FUNCTION_BLOCK ASSEMBLE_AL_FROM_AX (* this Function combines the 64 AX (BOOL) adapters to a AL (LWORD) *)
  (* Standard: 61499-2; Description: Copyright (c) 2026 Meisterschulen am Ostbahnhof SPDX-License-Identifier: EPL-2.0 *)
  (* Version 1.0, 2026-05-16, Franz Höpfinger, Meisterschulen am Ostbahnhof, initial API and implementation and/or initial documentation *)
  PACKAGE adapter::assembling;
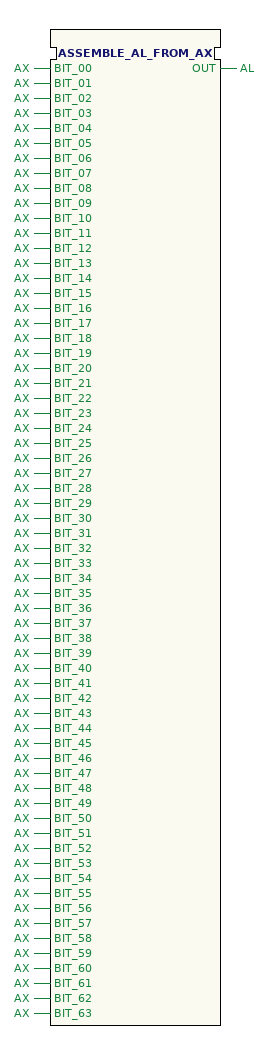
  SOCKETS
    BIT_00 : adapter::types::unidirectional::AX; (* Bool Bit 0 *)
    BIT_01 : adapter::types::unidirectional::AX; (* Bool Bit 1 *)
    BIT_02 : adapter::types::unidirectional::AX; (* Bool Bit 2 *)
    BIT_03 : adapter::types::unidirectional::AX; (* Bool Bit 3 *)
    BIT_04 : adapter::types::unidirectional::AX; (* Bool Bit 4 *)
    BIT_05 : adapter::types::unidirectional::AX; (* Bool Bit 5 *)
    BIT_06 : adapter::types::unidirectional::AX; (* Bool Bit 6 *)
    BIT_07 : adapter::types::unidirectional::AX; (* Bool Bit 7 *)
    BIT_08 : adapter::types::unidirectional::AX; (* Bool Bit 8 *)
    BIT_09 : adapter::types::unidirectional::AX; (* Bool Bit 9 *)
    BIT_10 : adapter::types::unidirectional::AX; (* Bool Bit 10 *)
    BIT_11 : adapter::types::unidirectional::AX; (* Bool Bit 11 *)
    BIT_12 : adapter::types::unidirectional::AX; (* Bool Bit 12 *)
    BIT_13 : adapter::types::unidirectional::AX; (* Bool Bit 13 *)
    BIT_14 : adapter::types::unidirectional::AX; (* Bool Bit 14 *)
    BIT_15 : adapter::types::unidirectional::AX; (* Bool Bit 15 *)
    BIT_16 : adapter::types::unidirectional::AX; (* Bool Bit 16 *)
    BIT_17 : adapter::types::unidirectional::AX; (* Bool Bit 17 *)
    BIT_18 : adapter::types::unidirectional::AX; (* Bool Bit 18 *)
    BIT_19 : adapter::types::unidirectional::AX; (* Bool Bit 19 *)
    BIT_20 : adapter::types::unidirectional::AX; (* Bool Bit 20 *)
    BIT_21 : adapter::types::unidirectional::AX; (* Bool Bit 21 *)
    BIT_22 : adapter::types::unidirectional::AX; (* Bool Bit 22 *)
    BIT_23 : adapter::types::unidirectional::AX; (* Bool Bit 23 *)
    BIT_24 : adapter::types::unidirectional::AX; (* Bool Bit 24 *)
    BIT_25 : adapter::types::unidirectional::AX; (* Bool Bit 25 *)
    BIT_26 : adapter::types::unidirectional::AX; (* Bool Bit 26 *)
    BIT_27 : adapter::types::unidirectional::AX; (* Bool Bit 27 *)
    BIT_28 : adapter::types::unidirectional::AX; (* Bool Bit 28 *)
    BIT_29 : adapter::types::unidirectional::AX; (* Bool Bit 29 *)
    BIT_30 : adapter::types::unidirectional::AX; (* Bool Bit 30 *)
    BIT_31 : adapter::types::unidirectional::AX; (* Bool Bit 31 *)
    BIT_32 : adapter::types::unidirectional::AX; (* Bool Bit 32 *)
    BIT_33 : adapter::types::unidirectional::AX; (* Bool Bit 33 *)
    BIT_34 : adapter::types::unidirectional::AX; (* Bool Bit 34 *)
    BIT_35 : adapter::types::unidirectional::AX; (* Bool Bit 35 *)
    BIT_36 : adapter::types::unidirectional::AX; (* Bool Bit 36 *)
    BIT_37 : adapter::types::unidirectional::AX; (* Bool Bit 37 *)
    BIT_38 : adapter::types::unidirectional::AX; (* Bool Bit 38 *)
    BIT_39 : adapter::types::unidirectional::AX; (* Bool Bit 39 *)
    BIT_40 : adapter::types::unidirectional::AX; (* Bool Bit 40 *)
    BIT_41 : adapter::types::unidirectional::AX; (* Bool Bit 41 *)
    BIT_42 : adapter::types::unidirectional::AX; (* Bool Bit 42 *)
    BIT_43 : adapter::types::unidirectional::AX; (* Bool Bit 43 *)
    BIT_44 : adapter::types::unidirectional::AX; (* Bool Bit 44 *)
    BIT_45 : adapter::types::unidirectional::AX; (* Bool Bit 45 *)
    BIT_46 : adapter::types::unidirectional::AX; (* Bool Bit 46 *)
    BIT_47 : adapter::types::unidirectional::AX; (* Bool Bit 47 *)
    BIT_48 : adapter::types::unidirectional::AX; (* Bool Bit 48 *)
    BIT_49 : adapter::types::unidirectional::AX; (* Bool Bit 49 *)
    BIT_50 : adapter::types::unidirectional::AX; (* Bool Bit 50 *)
    BIT_51 : adapter::types::unidirectional::AX; (* Bool Bit 51 *)
    BIT_52 : adapter::types::unidirectional::AX; (* Bool Bit 52 *)
    BIT_53 : adapter::types::unidirectional::AX; (* Bool Bit 53 *)
    BIT_54 : adapter::types::unidirectional::AX; (* Bool Bit 54 *)
    BIT_55 : adapter::types::unidirectional::AX; (* Bool Bit 55 *)
    BIT_56 : adapter::types::unidirectional::AX; (* Bool Bit 56 *)
    BIT_57 : adapter::types::unidirectional::AX; (* Bool Bit 57 *)
    BIT_58 : adapter::types::unidirectional::AX; (* Bool Bit 58 *)
    BIT_59 : adapter::types::unidirectional::AX; (* Bool Bit 59 *)
    BIT_60 : adapter::types::unidirectional::AX; (* Bool Bit 60 *)
    BIT_61 : adapter::types::unidirectional::AX; (* Bool Bit 61 *)
    BIT_62 : adapter::types::unidirectional::AX; (* Bool Bit 62 *)
    BIT_63 : adapter::types::unidirectional::AX; (* Bool Bit 63 *)
  END_SOCKETS
  PLUGS
    OUT : adapter::types::unidirectional::AL; (* LWORD Output *)
  END_PLUGS
END_FUNCTION_BLOCK
